Fanuc KAREL source: ko00016.KL

-- PROVISIONAL review KL for V1013-1; original PC SHA256 b3f5a6a21e231265b3c4c0cfb4867a0abe201b5e0f5d7edc726c8942fdfd1f24
-- Incomplete behavior may be omitted. Consult companion uncertainty JSON. Do not deploy.
PROGRAM KO00016
%NOLOCKGROUP
-- UNRESOLVED_DECL P1 type=000102
-- UNRESOLVED_DECL P2 type=000102
-- UNRESOLVED_DECL P3 type=000102
-- UNRESOLVED_DECL P4 type=000102
-- UNRESOLVED_DECL OUT type=000199
BEGIN
  -- UNRESOLVED_PC offsets 5-80; opcodes 27,27,49,7E,AD,27,49,7E,AD,27,49,7E,AD,27,49,7E,AD,76,7E,4A
  -- UNRESOLVED_PC offsets 85-89; opcodes 7F
END KO00016
